FUNCTION_BLOCK Skill_1
VAR_INPUT
	Var_1			:BOOL;
	Var_2			:BOOL;
END_VAR
VAR_OUTPUT
	
END_VAR
VAR
	Skill_1			:TestSkill;
END_VAR

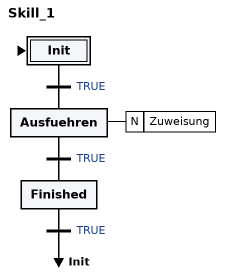
INITIAL_STEP Init:
END_STEP
TRANSITION FROM Init TO Ausfuehren
    := TRUE;
END_TRANSITION
STEP Ausfuehren:
    Zuweisung(N);
END_STEP
TRANSITION FROM Ausfuehren TO Finished
    := TRUE;
END_TRANSITION
STEP Finished:
END_STEP
TRANSITION FROM Finished TO Init
    := TRUE;
END_TRANSITION

ACTION Zuweisung:
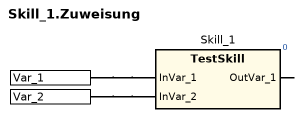
Skill_1(InVar_1 := Var_1, InVar_2 := Var_2); // TestSkill
END_ACTION

END_FUNCTION_BLOCK

(* stored: Version 1.1.0.1
   POU Skill_1: Id {234d6ee4-7cbc-4b59-bd9b-e34489ee7e39}, SpecialFunc None
   Action Zuweisung: Id {0cb60c39-3562-4b78-b409-99aec1b085b0} *)
